FUNCTION TryConvert_USINT_TO_DWORD : BOOL
VAR_INPUT
	in : USINT;
	out : REFERENCE TO DWORD;
END_VAR

out := USINT_TO_DWORD(in);
TryConvert_USINT_TO_DWORD := TRUE;

END_FUNCTION

(* stored: Version 1.1.0.1, ProductVersion 3.1.4024.12
   POU TryConvert_USINT_TO_DWORD: Id {62a1b683-6a11-45bc-9386-e47765d8e24f}, SpecialFunc None *)
